//EL7037 | Stepper motor terminal, 24V DC, 1.5A
FUNCTION_BLOCK EL7037

VAR_INPUT
    En: BOOL;
    iTerminal_ID : INT;
    ErrorSystem : POINTER TO ST_ErrorSystem;
END_VAR

VAR_OUTPUT
    EnO: BOOL;
    bError: BOOL;
END_VAR

VAR
    //WC_State is handled by NC, so NOT included here.
    InfoData_State AT %I*: UINT;

    //FB-s
    EL7037_Error    : FB_TerminalError;
END_VAR

(*
* TODO: Test on hardware
*)

EnO:=En;

EL7037_Error(
    En := TRUE,
    iTerminal_ID := iTerminal_ID,
    bWcState := FALSE,
    uiInfoData_State := InfoData_State,
    pErrorSystem := ErrorSystem,
    bError => bError,
);

END_FUNCTION_BLOCK

(* stored: Version 1.1.0.1, ProductVersion 3.1.4024.6
   POU EL7037: Id {27d5d25d-3c68-47ea-8be3-e1716776c522}, SpecialFunc None *)
